// TIA Portal V19 export
VAR_GLOBAL   // PLC tag table "conveyor-2"
   "Start Button 2-Left" AT %I0.3 : Bool;
   "Start Button 2-right" AT %I0.4 : Bool;
   "Stop Button 2" AT %I0.5 : Bool;
   "Belt Conveyor (4m) 2 (+)" AT %Q0.2 : Bool;
   "Belt Conveyor (4m) 2 (-)" AT %Q0.3 : Bool;
   "mem2-stop" AT %M2.2 : Bool;
   "mem-Belt Conveyor (4m) 2 (+)" AT %M2.3 : Bool;
   "mem-Belt Conveyor (4m) 2 (-)" AT %M2.4 : Bool;
   "mem-moment" AT %M2.5 : Bool;
END_VAR
